// TIA Portal V18 export
VAR_GLOBAL   // PLC tag table "04_4 Costanti Nomi Attuatore Stz04"
END_VAR
VAR_GLOBAL CONSTANT   // user constants
   M101 : Int := 1;   // Motore rotazione mandrino
   H401 : Int := 2;   // EV Espansione/contrazione mandrino
   H402 : Int := 3;   // EV Salita/discesa braccio premicoil
END_VAR
